FUNCTION_BLOCK I_WBSD (* Wheel-based Speed and Distance WBSD *)
  (* Standard: ISO 11783-7; Classification: PGN 65096; Function: Wheel-based Speed and Distance WBSD; Description: Copyright (c) 2024 HR Agrartechnik GmbH This program and the accompanying materials are made available under the terms of the Eclipse Public License 2.0 which is available at https://www.eclipse.org/legal/epl-2.0/ SPDX-License-Identifier: EPL-2.0 Message sent by the Tractor ECU on the implement bus on construction and agricultural implements providing to connected systems the current measured wheel-based speed. The message also includes a free-running distance counter, an indication of the direction of travel and the state of the start/stop switch or input. When the ignition key switch is turned off, both the ECU_PWR and PWR have to be maintained to send this message for an additional 2 s. This is not required when the engine is cranking (starting). Accuracies of both wheel-based and ground-based sources can be speed-dependent and degrade at low speeds. Wheel-based information might not be updated at the 100 ms rate at low speeds. https://docs.ms-muc-docs.de/projects/isobus-other-docs/de/latest/PGN/PGN_65096.html *)
  (* Version 1.0, 2024-07-09, Franz Höpfinger, HR Agrartechnik GmbH *)
  PACKAGE isobus::tecu;
  IMPORT eclipse4diac::core::TypeHash;
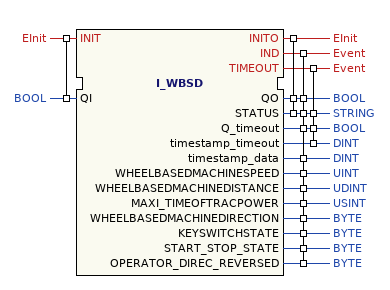
  EVENT_INPUT
    INIT : EInit WITH QI; (* Service Initialization *)
  END_EVENT
  EVENT_OUTPUT
    INITO : EInit WITH QO, STATUS; (* Initialization Confirm *)
    IND WITH QO, timestamp_data, WHEELBASEDMACHINESPEED, WHEELBASEDMACHINEDISTANCE, MAXI_TIMEOFTRACPOWER, WHEELBASEDMACHINEDIRECTION, KEYSWITCHSTATE, START_STOP_STATE, OPERATOR_DIREC_REVERSED, STATUS, Q_timeout; (* Indication from Resource *)
    TIMEOUT WITH timestamp_timeout, STATUS, Q_timeout;
  END_EVENT
  VAR_INPUT
    QI : BOOL; (* Event Input Qualifier *)
  END_VAR
  VAR_OUTPUT
    QO : BOOL; (* Event Output Qualifier *)
    STATUS : STRING;
    Q_timeout : BOOL;
    timestamp_timeout : DINT;
    timestamp_data : DINT;
    WHEELBASEDMACHINESPEED : UINT; (* Wheel-based machine speed (see Attributes for Details) *) {SET_ATTRIBUTE(SPN, 1862)} {SET_ATTRIBUTE(SP_Name, 'Wheel-based machine speed')} {SET_ATTRIBUTE(SP_Position_In_PG, '1-2')} {SET_ATTRIBUTE(SP_Length, 16)} (* 16 bits *) {SET_ATTRIBUTE(Scaling, '0.001 m/s per bit')} {SET_ATTRIBUTE(Offset, )} {SET_ATTRIBUTE(Link, 'https://docs.ms-muc-docs.de/projects/isobus-other-docs/de/latest/PGN/PGN_65096.html#spn-1862-wheel-based-machine-speed')}
    WHEELBASEDMACHINEDISTANCE : UDINT; (* Wheel-based machine distance (see Attributes for Details) *) {SET_ATTRIBUTE(SPN, 1863)} {SET_ATTRIBUTE(SP_Name, 'Wheel-based machine distance')} {SET_ATTRIBUTE(SP_Position_In_PG, '3-6')} {SET_ATTRIBUTE(SP_Length, 16)} (* 32 bits *) {SET_ATTRIBUTE(Scaling, '0.001 m/bit')} {SET_ATTRIBUTE(Offset, )} {SET_ATTRIBUTE(Link, 'https://docs.ms-muc-docs.de/projects/isobus-other-docs/de/latest/PGN/PGN_65096.html#spn-1863-wheel-based-machine-distance')}
    MAXI_TIMEOFTRACPOWER : USINT; (* Maximum Time of Tractor Power (see Attributes for Details) *) {SET_ATTRIBUTE(SPN, 1866)} {SET_ATTRIBUTE(SP_Name, 'Maximum Time of Tractor Power')} {SET_ATTRIBUTE(SP_Position_In_PG, '7')} {SET_ATTRIBUTE(SP_Length, 16)} (* 8 bits *) {SET_ATTRIBUTE(Scaling, '1 min/bit')} {SET_ATTRIBUTE(Offset, )} {SET_ATTRIBUTE(Link, 'https://docs.ms-muc-docs.de/projects/isobus-other-docs/de/latest/PGN/PGN_65096.html#spn-1866-maximum-time-of-tractor-power')}
    WHEELBASEDMACHINEDIRECTION : BYTE; (* Wheel-based machine direction (see Attributes for Details) *) {SET_ATTRIBUTE(SPN, 1864)} {SET_ATTRIBUTE(SP_Name, 'Wheel-based machine direction')} {SET_ATTRIBUTE(SP_Position_In_PG, '8.1')} {SET_ATTRIBUTE(SP_Length, 16)} (* 2 bits *) {SET_ATTRIBUTE(Scaling, '4 states/2 bit')} {SET_ATTRIBUTE(Offset, )} {SET_ATTRIBUTE(Link, 'https://docs.ms-muc-docs.de/projects/isobus-other-docs/de/latest/PGN/PGN_65096.html#spn-1864-wheel-based-machine-direction')}
    KEYSWITCHSTATE : BYTE; (* Key switch state (see Attributes for Details) *) {SET_ATTRIBUTE(SPN, 1865)} {SET_ATTRIBUTE(SP_Name, 'Key switch state')} {SET_ATTRIBUTE(SP_Position_In_PG, '8.3')} {SET_ATTRIBUTE(SP_Length, 16)} (* 2 bits *) {SET_ATTRIBUTE(Scaling, '4 states/2 bit')} {SET_ATTRIBUTE(Offset, )} {SET_ATTRIBUTE(Link, 'https://docs.ms-muc-docs.de/projects/isobus-other-docs/de/latest/PGN/PGN_65096.html#spn-1865-key-switch-state')}
    START_STOP_STATE : BYTE; (* Implement Start/Stop operations (see Attributes for Details) *) {SET_ATTRIBUTE(SPN, 5203)} {SET_ATTRIBUTE(SP_Name, 'Implement Start/Stop operations')} {SET_ATTRIBUTE(SP_Position_In_PG, '8.5')} {SET_ATTRIBUTE(SP_Length, 16)} (* 2 bits *) {SET_ATTRIBUTE(Scaling, '4 states/2 bit')} {SET_ATTRIBUTE(Offset, )} {SET_ATTRIBUTE(Link, 'https://docs.ms-muc-docs.de/projects/isobus-other-docs/de/latest/PGN/PGN_65096.html#spn-5203-implement-start-stop-operations')}
    OPERATOR_DIREC_REVERSED : BYTE; (* Operator direction reversed (see Attributes for Details) *) {SET_ATTRIBUTE(SPN, 5244)} {SET_ATTRIBUTE(SP_Name, 'Operator direction reversed')} {SET_ATTRIBUTE(SP_Position_In_PG, '8.7')} {SET_ATTRIBUTE(SP_Length, 16)} (* 2 bits *) {SET_ATTRIBUTE(Scaling, '4 states/2 bit')} {SET_ATTRIBUTE(Offset, )} {SET_ATTRIBUTE(Link, 'https://docs.ms-muc-docs.de/projects/isobus-other-docs/de/latest/PGN/PGN_65096.html#spn-5244-operator-direction-reversed')}
  END_VAR
END_FUNCTION_BLOCK
